INTERFACE I_FillingStrategy

METHOD ExecuteFill : BOOL
VAR_INPUT
	stBottle : REFERENCE TO ST_Bottle;
END_VAR
END_METHOD

END_INTERFACE

(* stored: Version 1.1.0.1, ProductVersion 3.1.4024.16
   Itf I_FillingStrategy: Id {519cdf10-2323-421f-84b3-4f02b8705776}
   Method ExecuteFill: Id {db11ecaa-1951-495f-a7e4-c8be23aae2e1} *)
